// TwinCAT 3 PLC project PLC
// ProgramVersion: 3.1.4026.19
// libraries:
//   SPT Base Types, * (Beckhoff Automation LLC)
//   SPT Components, * (Beckhoff Automation LLC)
//   SPT Diagnostic, * (Beckhoff Automation LLC)
//   SPT EtherCat, * (Beckhoff Automation LLC)
//   SPT Event Logger, * (Beckhoff Automation LLC)
//   SPT Motion Control, * (Beckhoff Automation LLC)
//   SPT Utilities, * (Beckhoff Automation LLC)
//   Tc2_MC2, * (Beckhoff Automation GmbH)
//   Tc2_MC2_Camming, * (Beckhoff Automation GmbH)
//   Tc2_Standard, * (Beckhoff Automation GmbH)
//   Tc2_System, * (Beckhoff Automation GmbH)
//   Tc3_EventLogger, * (Beckhoff Automation GmbH)
//   Tc3_Module, * (Beckhoff Automation GmbH)
//   Tc3_PackML_V3, * (Beckhoff Automation GmbH)
// project tree:
//   / GlobalTextList.TcGTLO, PlcTask.TcTTO, Visualization Manager.TcVMO (not stored)
//   Modules/00 Machine/ Machine.TcPOU
//   Modules/01 Cam Module Table Select/ CamModule_TableSelect.TcPOU
//   Modules/01 Cam Module Table Select/DUTs/ ST_EM_Cfg_TableSelect.TcDUT, ST_EM_Cmd_TableSelect.TcDUT, ST_EM_HMI_TableSelect.TcDUT, ST_EM_Sts_TableSelect.TcDUT
//   Modules/02 Cam Module Update Table/ CamModule_UpdateTable.TcPOU
//   Modules/02 Cam Module Update Table/DUTs/ ST_EM_Cfg_UpdateTable.TcDUT, ST_EM_Cmd_UpdateTable.TcDUT, ST_EM_HMI_UpdateTable.TcDUT, ST_EM_Sts_UpdateTable.TcDUT
//   POUs/ MAIN.TcPOU
//   VISUs/ Visualization.TcVIS
// real-time tasks:
//   TASK PlcTask: cycle T#10ms, priority 20, ADS port 350
// motion (NC):
//   TASK NC-Task 1 SAF: cycle T#2ms, priority 4, ADS port 501
//   TASK NC-Task 1 SVB: cycle T#10ms, priority 8, ADS port 511
//   AXIS Cam Shaft Table Select (id 1)
//     OtherSettings: AllowMotionCmdToSlave=true
//     encoder EncType=1
//     drive DrvType=5
//       Analog: TorqueSetpointScale=10, ScaleFactorActTorque=0.1
//       TimeComp: TaskDelayCycles=1
//     controller CtrType=1
//       CtrPara: PriorControlFactor=1
//         Observer: BandWidth=20
//   AXIS Cam Follower Table Select (id 2)
//     OtherSettings: AllowMotionCmdToSlave=true
//     encoder EncType=1
//     drive DrvType=5
//       Analog: TorqueSetpointScale=10, ScaleFactorActTorque=0.1
//       TimeComp: TaskDelayCycles=1
//     controller CtrType=1
//       CtrPara: PriorControlFactor=1
//         Observer: BandWidth=20
//   AXIS Cam Shaft Update Table (id 3)
//     General: UnitFlags=#x00000004
//     OtherSettings: AllowMotionCmdToSlave=true
//     encoder EncType=1
//     drive DrvType=5
//       Analog: TorqueSetpointScale=10, ScaleFactorActTorque=0.1
//       TimeComp: TaskDelayCycles=1
//     controller CtrType=1
//       CtrPara: PriorControlFactor=1
//         Observer: BandWidth=20
//   AXIS Cam Follwer Update Table (id 4)
//     OtherSettings: AllowMotionCmdToSlave=true
//     encoder EncType=1
//     drive DrvType=5
//       Analog: TorqueSetpointScale=10, ScaleFactorActTorque=0.1
//     controller CtrType=1
//       CtrPara: PriorControlFactor=1
//         Observer: BandWidth=20
// variable links:
//   PLC/PLC Instance <-> NC-Task 1 SAF/Axes/Cam Follower Table Select
//     PlcTask Inputs/MAIN.Machine.CamModule_TableSelect.CamFollower.CamSlaveAxis._Axis.NcToPlc <-> Outputs/ToPlc
//     PlcTask Outputs/MAIN.Machine.CamModule_TableSelect.CamFollower.CamSlaveAxis._Axis.PlcToNc <-> Inputs/FromPlc
//   PLC/PLC Instance <-> NC-Task 1 SAF/Axes/Cam Follwer Update Table
//     PlcTask Inputs/MAIN.Machine.CamModule_UpdateTable.CamFollower.CamSlaveAxis._Axis.NcToPlc <-> Outputs/ToPlc
//     PlcTask Outputs/MAIN.Machine.CamModule_UpdateTable.CamFollower.CamSlaveAxis._Axis.PlcToNc <-> Inputs/FromPlc
//   PLC/PLC Instance <-> NC-Task 1 SAF/Axes/Cam Shaft Table Select
//     PlcTask Inputs/MAIN.Machine.CamModule_TableSelect.CamShaft.BasicAxis._Axis.NcToPlc <-> Outputs/ToPlc
//     PlcTask Outputs/MAIN.Machine.CamModule_TableSelect.CamShaft.BasicAxis._Axis.PlcToNc <-> Inputs/FromPlc
//   PLC/PLC Instance <-> NC-Task 1 SAF/Axes/Cam Shaft Update Table
//     PlcTask Inputs/MAIN.Machine.CamModule_UpdateTable.CamShaft.BasicAxis._Axis.NcToPlc <-> Outputs/ToPlc
//     PlcTask Outputs/MAIN.Machine.CamModule_UpdateTable.CamShaft.BasicAxis._Axis.PlcToNc <-> Inputs/FromPlc

CONFIGURATION PLC
    RESOURCE PLC ON TwinCAT3
        TASK PlcTask(INTERVAL := T#10ms, PRIORITY := 20);
        PROGRAM MAIN WITH PlcTask : MAIN;
    END_RESOURCE
END_CONFIGURATION

// ---- Modules/01 Cam Module Table Select/DUTs/ST_EM_Cfg_TableSelect.TcDUT
TYPE ST_EM_Cfg_TableSelect :
	STRUCT
		CamActivationMode : INT;
	END_STRUCT
END_TYPE

// ---- Modules/01 Cam Module Table Select/DUTs/ST_EM_Cmd_TableSelect.TcDUT
TYPE ST_EM_Cmd_TableSelect :
	STRUCT
		ChangeTable : BOOL;
		ChangeMode	: BOOL;
	END_STRUCT
END_TYPE

// ---- Modules/01 Cam Module Table Select/DUTs/ST_EM_HMI_TableSelect.TcDUT
TYPE ST_EM_HMI_TableSelect :
	STRUCT
		Cmd : ST_EM_Cmd_TableSelect;
		Cfg : ST_EM_Cfg_TableSelect;
		Sts : ST_EM_Sts_TableSelect;
	END_STRUCT
END_TYPE

// ---- Modules/01 Cam Module Table Select/DUTs/ST_EM_Sts_TableSelect.TcDUT
TYPE ST_EM_Sts_TableSelect :
	STRUCT
		CurrentTable : UDINT;
	END_STRUCT
END_TYPE

// ---- Modules/02 Cam Module Update Table/DUTs/ST_EM_Cfg_UpdateTable.TcDUT
TYPE ST_EM_Cfg_UpdateTable :
	STRUCT
		CamActivationMode : INT;
	END_STRUCT
END_TYPE

// ---- Modules/02 Cam Module Update Table/DUTs/ST_EM_Cmd_UpdateTable.TcDUT
TYPE ST_EM_Cmd_UpdateTable :
	STRUCT
		ChangeTable : BOOL;
		ChangeMode	: BOOL;
	END_STRUCT
END_TYPE

// ---- Modules/02 Cam Module Update Table/DUTs/ST_EM_HMI_UpdateTable.TcDUT
TYPE ST_EM_HMI_UpdateTable :
	STRUCT
		Cmd : ST_EM_Cmd_UpdateTable;
		Cfg : ST_EM_Cfg_UpdateTable;
		Sts : ST_EM_Sts_UpdateTable;
	END_STRUCT
END_TYPE

// ---- Modules/02 Cam Module Update Table/DUTs/ST_EM_Sts_UpdateTable.TcDUT
TYPE ST_EM_Sts_UpdateTable :
	STRUCT
		CurrentTable : UDINT;
	END_STRUCT
END_TYPE

// ---- POUs/MAIN.TcPOU
PROGRAM MAIN
VAR
	Machine : Machine := (Name := 'Machine');
END_VAR

// All sample code provided by Beckhoff Automation LLC are for illustrative purposes only and are provided “as is” and without any warranties, express or implied. Actual implementations in applications will vary significantly. Beckhoff Automation LLC shall have no liability for, and does not waive any rights in relation to, any code samples that it provides or the use of such code samples for any purpose.

(*
	Each Equipment Module holds 2 Axes.
	The first is the Cam Shaft (Master Axis), and the second is the Cam Follwer that will follow the cam table as the Cam Shaft is mmoving.
	The Cam table data is first populated during the Initialize method.

	The default value for ActivationMode is MC_CAMACTIVATION_INSTANTANEOUS.
	In the Cyclic Logic method the ActivationMode can be changed to:
	MC_CamActivationMode.MC_CAMACTIVATION_INSTANTANEOUS
	MC_CamActivationMode.MC_CAMACTIVATION_NEXTCYCLE
	MC_CamActivationMode.MC_CAMACTIVATION_ASSOONASPOSSIBLE
	
	Cam Module Table Select creates 2 tables in the Initialize method.
	Table 1 and Table 2
	In the Execute method it is possible to switch between tables based on the ActivationMode.
	
	Cam Module Update Table creates a single table in the Initialize method.
	In the Execute method the TableID is changed, the WriteParameters_1 or _2 is called to populate the new data, and the the UpdateTable() method is called.
	This process will continue to use the same table, but use the new values provided.

	The Visu provides the functionality to update the the running table based on the tables defined within the CamParameters.CamTable array.


*)

// For Debug Only
_AppInfo.KeepOutputsOnBP := TRUE;

//
Machine.CyclicLogic();

END_PROGRAM

// ---- Modules/00 Machine/Machine.TcPOU
FUNCTION_BLOCK Machine EXTENDS FB_PackML_BaseModule
VAR
	CamModule_TableSelect : CamModule_TableSelect := (Name := 'Cam Module Table Select');
	CamModule_UpdateTable : CamModule_UpdateTable := (Name := 'Cam Module Update Table');
END_VAR

// Automatically enables and disables HMI control based on the PackML mode
METHOD PROTECTED HMIPermissions

// This method is called cyclically by CyclicLogic()
AllowHMIControl(TRUE);
END_METHOD

// Basic module initialization logic
METHOD PROTECTED Initialize : BOOL;

// This method is called by CyclicLogic() as required
Initialize := FALSE;
CASE DescendantSequenceState OF
	0:
		RegisterSubmodule(SubModule := CamModule_TableSelect);
		RegisterSubmodule(SubModule := CamModule_UpdateTable);
		DescendantSequenceState := DescendantSequenceState + 10;

	10:
		IF SUPER^.Initialize() THEN
			Initialize := TRUE;
		END_IF
END_CASE
END_METHOD

END_FUNCTION_BLOCK

// ---- Modules/01 Cam Module Table Select/CamModule_TableSelect.TcPOU
FUNCTION_BLOCK CamModule_TableSelect EXTENDS FB_PackML_BaseModule
VAR
	CamShaft	  : FB_Component_BasicAxis	  := (Name := 'Cam Shaft');
	CamFollower	  : FB_Component_CamSlaveAxis := (Name := 'Cam Follower');
	CamParameters : ST_CamParameters;
	HMI			  : ST_EM_HMI_TableSelect;
END_VAR

METHOD PROTECTED Aborting
VAR
	CamShaftStop	: BOOL;
	CamFollowerStop : BOOL;
END_VAR
// Mode is ignored
CASE SequenceState OF
	0:
		NoStateTasksToComplete := FALSE;
		SequenceState		   := SequenceState + 10;

		// Setting Override to 100 will ensure velocity calculations are not limited
		CamShaft.Override	 := 100;
		CamFollower.Override := 100;

		// The below code is used to call the stop method of each axis while still in State 0, this is done for efficeniceny while aborting.

		// Stop all Axes
		CamShaftStop	:= CamShaft.Stop() OR CamShaft.Error;
		CamFollowerStop := CamFollower.Stop() OR CamFollower.Error;
		IF CamShaftStop AND CamFollowerStop THEN
			SequenceState := SequenceState + 10;
		END_IF

	10:
		IF CamShaft.Stopped AND CamFollower.Stopped THEN
			SequenceState := SequenceState + 10;
		END_IF

	20: // Disable Axis
		IF CamShaft.Disable() THEN
			SequenceState := SequenceState + 10;
		END_IF

	30:
		IF CamFollower.Disable() THEN
			SequenceState := SequenceState + 10;
		END_IF

	40:
		IF NOT CamShaft.Enabled AND NOT CamFollower.Enabled THEN
			SequenceState := SequenceState + 10;
		END_IF

	50:
		StateTasksComplete := TRUE;
END_CASE

SUPER^.Aborting();
END_METHOD

// This method contains code which will execute when this PackML module is in the Clearing state
METHOD PROTECTED Clearing

// Note: The Clear command can also be thought of as a fault reset depite the ambiguity in the naming of the Reset state. 

// This method is called as required by StateControl()
// Mode is ignored
CASE SequenceState OF
	0:
		NoStateTasksToComplete := FALSE;
		SequenceState		   := SequenceState + 10;

	10: // Reset Axis if Error
		IF CamShaft.Error THEN
			IF CamShaft.Reset() THEN
				SequenceState := SequenceState + 10;
			END_IF
		ELSE
			SequenceState := SequenceState + 10;
		END_IF

	20:
		IF CamFollower.InSync THEN
			IF CamFollower.Stop() THEN // This is used to decouple the axis
				SequenceState := SequenceState + 10;
			END_IF
		ELSE
			SequenceState := SequenceState + 10;
		END_IF

	30:
		IF CamFollower.Error THEN
			IF CamFollower.Reset() THEN
				SequenceState := SequenceState + 10;
			END_IF
		ELSE
			SequenceState := SequenceState + 10;
		END_IF

	40:
		StateTasksComplete := TRUE;
END_CASE

SUPER^.Clearing();
END_METHOD

METHOD PROTECTED Completing
CASE SequenceState OF
	0:
		NoStateTasksToComplete := FALSE;
		SequenceState		   := SequenceState + 10;

	10:
		IF CamShaft.Stop() THEN // This will also GearOut
			SequenceState := SequenceState + 10;
		END_IF

	20:
		IF CamFollower.Stop() THEN // This will also GearOut
			SequenceState := SequenceState + 10;
		END_IF

	30:
		IF CamShaft.Stopped AND CamFollower.Stopped THEN
			SequenceState := SequenceState + 10;
		END_IF

	40:
		StateTasksComplete := TRUE;
END_CASE

SUPER^.Completing();
END_METHOD

// This method serves as the entry point for all underlying FB logic

// This method should be called cyclically by descendant function blocks by invoking SUPER^.CyclicLogic().  Alternatively, the contents of this method could be reimplemented entirely in which case a call to this method would not be necessary.
METHOD PUBLIC CyclicLogic
IF NOT _InitComplete THEN
	_InitComplete := Initialize();
	RETURN;
END_IF

// HMI Status Update
HMI.Sts.CurrentTable := CamFollower.RunningTable;

// Change Activation Mode
IF HMI.Cmd.ChangeMode THEN
	CASE HMI.Cfg.CamActivationMode OF
		0:
			CamParameters.ChangeOptions.ActivationMode := MC_CamActivationMode.MC_CAMACTIVATION_INSTANTANEOUS;

		1:
			CamParameters.ChangeOptions.ActivationMode := MC_CamActivationMode.MC_CAMACTIVATION_NEXTCYCLE;

		2:
			CamParameters.ChangeOptions.ActivationMode := MC_CamActivationMode.MC_CAMACTIVATION_ASSOONASPOSSIBLE;
	END_CASE

	IF CamFollower.ChangeMode() THEN
		HMI.Cmd.ChangeMode := FALSE;
	END_IF
END_IF

SUPER^.CyclicLogic();
END_METHOD

// This method contains code which will execute when this PackML module is in the Execute state
METHOD PROTECTED Execute

(*
The base implementation of this method is empty. User must override this method to provide functionality.
This method is called as required by StateControl()
*)
CASE _CurrentMode OF
	E_PMLUnitMode.Production:
		CASE SequenceState OF
			0: // Start Cam Shaft
				IF CamShaft.MoveVelocity(50.0, FALSE) THEN
					SequenceState := SequenceState + 10;
				END_IF

			10: // Checking that the Cam Shaft is near the commanded speed 
				IF (CamShaft.ActualVelocity > (CamShaft.SetVelocity * 0.9)) THEN
					SequenceState := SequenceState + 10;
				END_IF

			20:
				IF HMI.Cmd.ChangeTable THEN
					HMI.Cmd.ChangeTable := FALSE;
					CASE CamFollower.RunningTable OF
						1:
							CamFollower.CamParameters.TableSelect := 2;

						2:
							CamFollower.CamParameters.TableSelect := 1;
					END_CASE

					SequenceState := SequenceState + 10;
				END_IF

			30:
				IF CamFollower.RunningTable = CamFollower.CamParameters.TableSelect THEN
					SequenceState := 20;
				END_IF;
		END_CASE
END_CASE
END_METHOD

// Basic module initialization logic
METHOD PROTECTED Initialize : BOOL;

// This method is called by CyclicLogic() as required
Initialize := FALSE;
CASE DescendantSequenceState OF
	0:
		RegisterComponent(Component := CamShaft);
		RegisterComponent(Component := CamFollower);
		DescendantSequenceState := DescendantSequenceState + 10;

	10:
		IF SUPER^.Initialize() THEN
			DescendantSequenceState := DescendantSequenceState + 10;
		END_IF

	20:
		// Create the Cam table data and store in CamParameters
		WriteCamParameters();

		// Set the Reference for the Axis Cam Parameters to the CamParameters
		CamFollower.CamParameters REF= CamParameters;

		// Setting the Reference of the FB_Component_CamSlaveAxis must be done after the component has been initialized
		CamFollower.Master REF= CamShaft.Axis;

		//
		DescendantSequenceState := DescendantSequenceState + 10;

	30:
		Initialize := TRUE;
END_CASE
END_METHOD

METHOD PROTECTED Starting
CASE _CommandedMode OF
	E_PMLUnitMode.Production:
		CASE SequenceState OF
			0:
				NoStateTasksToComplete := FALSE;
				SequenceState		   := SequenceState + 10;

			10: // Enable Axis 
				IF CamShaft.Enable() THEN
					SequenceState := SequenceState + 10;
				END_IF

			20:
				IF CamShaft.Enabled THEN
					SequenceState := SequenceState + 10;
				END_IF

			30: // This step is not required, but is used in this demo to ensure the CamShaft starts at 0
				IF CamShaft.MoveModulo(0.0, MC_Direction.MC_Shortest_Way, 0) THEN
					SequenceState := SequenceState + 10;
				END_IF

			40:
				IF NOT CamShaft.Busy THEN
					IF NOT CamShaft.Error THEN
						SequenceState := SequenceState + 10;
					END_IF
				END_IF

			50: // Enable Axis
				IF CamFollower.Enable() THEN
					SequenceState := SequenceState + 10;
				END_IF

			60:
				IF CamFollower.Enabled THEN
					SequenceState := SequenceState + 10;
				END_IF

			70: // This step is not required, but is used in the demo to ensure the follower starts at 0
				IF CamFollower.MoveAbsolute(0, 0) THEN
					SequenceState := SequenceState + 10;
				END_IF

			80:
				IF NOT CamFollower.Busy THEN
					IF NOT CamFollower.Error THEN
						SequenceState := SequenceState + 10;
					END_IF
				END_IF

			90: // Verify the Master axis is ready 
				IF CamFollower.Master.Status.Operational THEN
					SequenceState := SequenceState + 10;
				END_IF

			100: // Select the Cam Table to be used
				CamFollower.CamParameters.TableSelect := 1;
				SequenceState						  := SequenceState + 10;

			110: // Couple to Cam table with Master axis
				IF CamFollower.WaitingForCommand THEN
					IF CamFollower.StartSync() THEN // The Start Sync command will move the axes tho the necessary positions and then CamIn
						SequenceState := SequenceState + 10;
					END_IF
				END_IF

			120:
				IF CamFollower.InSync THEN
					SequenceState := SequenceState + 10;
				END_IF

			130:
				StateTasksComplete := TRUE;
		END_CASE
END_CASE

SUPER^.Starting();
END_METHOD

METHOD PROTECTED Stopping
CASE SequenceState OF
	0:
		NoStateTasksToComplete := FALSE;
		SequenceState		   := SequenceState + 10;

	10:
		IF CamShaft.Stop() THEN // This will also GearOut 
			SequenceState := SequenceState + 10;
		END_IF

	20:
		IF CamFollower.Stop() THEN // This will also GearOut  
			SequenceState := SequenceState + 10;
		END_IF

	30:
		IF CamShaft.Stopped AND CamFollower.Stopped THEN
			SequenceState := SequenceState + 10;
		END_IF

	40:
		StateTasksComplete := TRUE;
END_CASE

SUPER^.Stopping();
END_METHOD

METHOD WriteCamParameters
VAR
	PointIdx : UDINT;
	i		 : UDINT;
	Start	 : UDINT;
END_VAR
// Table 1 Data
CamParameters.CamTableId										:= CamShaft.Axis.NcToPlc.AxisId;
CamParameters.CamTable[CamParameters.CamTableId].NumberOfPoints := Parameters_MotionControl.CAM_SLAVE_AXIS_MAX_CAM_POINTS;
PointIdx														:= 0;

//
PointIdx																			:= PointIdx + 1;
CamParameters.CamTable[CamParameters.CamTableId].Points[PointIdx].PointIndex		:= PointIdx;
CamParameters.CamTable[CamParameters.CamTableId].Points[PointIdx].FunctionType		:= MC_MotionFunctionType.MOTIONFUNCTYPE_POLYNOM5;
CamParameters.CamTable[CamParameters.CamTableId].Points[PointIdx].PointType			:= MC_MotionPointType.MOTIONPOINTTYPE_REST;
CamParameters.CamTable[CamParameters.CamTableId].Points[PointIdx].RelIndexNextPoint := 1;
CamParameters.CamTable[CamParameters.CamTableId].Points[PointIdx].MasterPos			:= 0.0;
CamParameters.CamTable[CamParameters.CamTableId].Points[PointIdx].SlavePos			:= 0.0;

//
PointIdx																			:= PointIdx + 1;
CamParameters.CamTable[CamParameters.CamTableId].Points[PointIdx].PointIndex		:= PointIdx;
CamParameters.CamTable[CamParameters.CamTableId].Points[PointIdx].FunctionType		:= MC_MotionFunctionType.MOTIONFUNCTYPE_POLYNOM5;
CamParameters.CamTable[CamParameters.CamTableId].Points[PointIdx].PointType			:= MC_MotionPointType.MOTIONPOINTTYPE_VELOCITY;
CamParameters.CamTable[CamParameters.CamTableId].Points[PointIdx].RelIndexNextPoint := 1;
CamParameters.CamTable[CamParameters.CamTableId].Points[PointIdx].MasterPos			:= 90.0;
CamParameters.CamTable[CamParameters.CamTableId].Points[PointIdx].SlavePos			:= 0.0;

//
PointIdx																			:= PointIdx + 1;
CamParameters.CamTable[CamParameters.CamTableId].Points[PointIdx].PointIndex		:= PointIdx;
CamParameters.CamTable[CamParameters.CamTableId].Points[PointIdx].FunctionType		:= MC_MotionFunctionType.MOTIONFUNCTYPE_POLYNOM5;
CamParameters.CamTable[CamParameters.CamTableId].Points[PointIdx].PointType			:= MC_MotionPointType.MOTIONPOINTTYPE_VELOCITY;
CamParameters.CamTable[CamParameters.CamTableId].Points[PointIdx].RelIndexNextPoint := 1;
CamParameters.CamTable[CamParameters.CamTableId].Points[PointIdx].MasterPos			:= 180.0;
CamParameters.CamTable[CamParameters.CamTableId].Points[PointIdx].SlavePos			:= 10.0;

//
PointIdx																			:= PointIdx + 1;
CamParameters.CamTable[CamParameters.CamTableId].Points[PointIdx].PointIndex		:= PointIdx;
CamParameters.CamTable[CamParameters.CamTableId].Points[PointIdx].FunctionType		:= MC_MotionFunctionType.MOTIONFUNCTYPE_POLYNOM5;
CamParameters.CamTable[CamParameters.CamTableId].Points[PointIdx].PointType			:= MC_MotionPointType.MOTIONPOINTTYPE_VELOCITY;
CamParameters.CamTable[CamParameters.CamTableId].Points[PointIdx].RelIndexNextPoint := 1;
CamParameters.CamTable[CamParameters.CamTableId].Points[PointIdx].MasterPos			:= 270.0;
CamParameters.CamTable[CamParameters.CamTableId].Points[PointIdx].SlavePos			:= 10.0;

//
PointIdx																			:= PointIdx + 1;
CamParameters.CamTable[CamParameters.CamTableId].Points[PointIdx].PointIndex		:= PointIdx;
CamParameters.CamTable[CamParameters.CamTableId].Points[PointIdx].FunctionType		:= MC_MotionFunctionType.MOTIONFUNCTYPE_POLYNOM5;
CamParameters.CamTable[CamParameters.CamTableId].Points[PointIdx].PointType			:= MC_MotionPointType.MOTIONPOINTTYPE_VELOCITY;
CamParameters.CamTable[CamParameters.CamTableId].Points[PointIdx].RelIndexNextPoint := 1;
CamParameters.CamTable[CamParameters.CamTableId].Points[PointIdx].MasterPos			:= 360.0;
CamParameters.CamTable[CamParameters.CamTableId].Points[PointIdx].SlavePos			:= 0.0;

// Fill the rest of the table with ignore points
Start := PointIdx + 1;
FOR PointIdx := Start TO Parameters_MotionControl.CAM_SLAVE_AXIS_MAX_CAM_POINTS DO
	CamParameters.CamTable[CamParameters.CamTableId].Points[PointIdx].PointIndex		:= PointIdx;
	CamParameters.CamTable[CamParameters.CamTableId].Points[PointIdx].FunctionType		:= MC_MotionFunctionType.MOTIONFUNCTYPE_NOTDEF;
	CamParameters.CamTable[CamParameters.CamTableId].Points[PointIdx].PointType			:= MC_MotionPointType.MOTIONPOINTTYPE_IGNORE;
	CamParameters.CamTable[CamParameters.CamTableId].Points[PointIdx].RelIndexNextPoint := 1;
	CamParameters.CamTable[CamParameters.CamTableId].Points[PointIdx].MasterPos			:= 0.0;
	CamParameters.CamTable[CamParameters.CamTableId].Points[PointIdx].SlavePos			:= 0.0;
END_FOR

// Set Lasst Point RelNext to 0
CamParameters.CamTable[CamParameters.CamTableId].Points[Parameters_MotionControl.CAM_SLAVE_AXIS_MAX_CAM_POINTS].RelIndexNextPoint := 0;

// Table 2 Data
CamParameters.CamTableId										:= CamShaft.Axis.NcToPlc.AxisId + 1;
CamParameters.CamTable[CamParameters.CamTableId].NumberOfPoints := Parameters_MotionControl.CAM_SLAVE_AXIS_MAX_CAM_POINTS;
PointIdx														:= 0;

//
PointIdx																			:= PointIdx + 1;
CamParameters.CamTable[CamParameters.CamTableId].Points[PointIdx].PointIndex		:= PointIdx;
CamParameters.CamTable[CamParameters.CamTableId].Points[PointIdx].FunctionType		:= MC_MotionFunctionType.MOTIONFUNCTYPE_POLYNOM5;
CamParameters.CamTable[CamParameters.CamTableId].Points[PointIdx].PointType			:= MC_MotionPointType.MOTIONPOINTTYPE_REST;
CamParameters.CamTable[CamParameters.CamTableId].Points[PointIdx].RelIndexNextPoint := 1;
CamParameters.CamTable[CamParameters.CamTableId].Points[PointIdx].MasterPos			:= 0.0;
CamParameters.CamTable[CamParameters.CamTableId].Points[PointIdx].SlavePos			:= 0.0;

//
PointIdx																			:= PointIdx + 1;
CamParameters.CamTable[CamParameters.CamTableId].Points[PointIdx].PointIndex		:= PointIdx;
CamParameters.CamTable[CamParameters.CamTableId].Points[PointIdx].FunctionType		:= MC_MotionFunctionType.MOTIONFUNCTYPE_POLYNOM5;
CamParameters.CamTable[CamParameters.CamTableId].Points[PointIdx].PointType			:= MC_MotionPointType.MOTIONPOINTTYPE_VELOCITY;
CamParameters.CamTable[CamParameters.CamTableId].Points[PointIdx].RelIndexNextPoint := 1;
CamParameters.CamTable[CamParameters.CamTableId].Points[PointIdx].MasterPos			:= 90.0;
CamParameters.CamTable[CamParameters.CamTableId].Points[PointIdx].SlavePos			:= 0.0;

//
PointIdx																			:= PointIdx + 1;
CamParameters.CamTable[CamParameters.CamTableId].Points[PointIdx].PointIndex		:= PointIdx;
CamParameters.CamTable[CamParameters.CamTableId].Points[PointIdx].FunctionType		:= MC_MotionFunctionType.MOTIONFUNCTYPE_POLYNOM5;
CamParameters.CamTable[CamParameters.CamTableId].Points[PointIdx].PointType			:= MC_MotionPointType.MOTIONPOINTTYPE_VELOCITY;
CamParameters.CamTable[CamParameters.CamTableId].Points[PointIdx].RelIndexNextPoint := 1;
CamParameters.CamTable[CamParameters.CamTableId].Points[PointIdx].MasterPos			:= 180.0;
CamParameters.CamTable[CamParameters.CamTableId].Points[PointIdx].SlavePos			:= 20.0;

//
PointIdx																			:= PointIdx + 1;
CamParameters.CamTable[CamParameters.CamTableId].Points[PointIdx].PointIndex		:= PointIdx;
CamParameters.CamTable[CamParameters.CamTableId].Points[PointIdx].FunctionType		:= MC_MotionFunctionType.MOTIONFUNCTYPE_POLYNOM5;
CamParameters.CamTable[CamParameters.CamTableId].Points[PointIdx].PointType			:= MC_MotionPointType.MOTIONPOINTTYPE_REST;
CamParameters.CamTable[CamParameters.CamTableId].Points[PointIdx].RelIndexNextPoint := 1;
CamParameters.CamTable[CamParameters.CamTableId].Points[PointIdx].MasterPos			:= 270.0;
CamParameters.CamTable[CamParameters.CamTableId].Points[PointIdx].SlavePos			:= 20.0;

//
PointIdx																			:= PointIdx + 1;
CamParameters.CamTable[CamParameters.CamTableId].Points[PointIdx].PointIndex		:= PointIdx;
CamParameters.CamTable[CamParameters.CamTableId].Points[PointIdx].FunctionType		:= MC_MotionFunctionType.MOTIONFUNCTYPE_POLYNOM5;
CamParameters.CamTable[CamParameters.CamTableId].Points[PointIdx].PointType			:= MC_MotionPointType.MOTIONPOINTTYPE_REST;
CamParameters.CamTable[CamParameters.CamTableId].Points[PointIdx].RelIndexNextPoint := 1;
CamParameters.CamTable[CamParameters.CamTableId].Points[PointIdx].MasterPos			:= 360.0;
CamParameters.CamTable[CamParameters.CamTableId].Points[PointIdx].SlavePos			:= 0.0;

// Fill the rest of the table with ignore points
Start := PointIdx + 1;
FOR PointIdx := Start TO Parameters_MotionControl.CAM_SLAVE_AXIS_MAX_CAM_POINTS DO
	CamParameters.CamTable[CamParameters.CamTableId].Points[PointIdx].PointIndex		:= PointIdx;
	CamParameters.CamTable[CamParameters.CamTableId].Points[PointIdx].FunctionType		:= MC_MotionFunctionType.MOTIONFUNCTYPE_NOTDEF;
	CamParameters.CamTable[CamParameters.CamTableId].Points[PointIdx].PointType			:= MC_MotionPointType.MOTIONPOINTTYPE_IGNORE;
	CamParameters.CamTable[CamParameters.CamTableId].Points[PointIdx].RelIndexNextPoint := 1;
	CamParameters.CamTable[CamParameters.CamTableId].Points[PointIdx].MasterPos			:= 0.0;
	CamParameters.CamTable[CamParameters.CamTableId].Points[PointIdx].SlavePos			:= 0.0;
END_FOR

// Set Lasst Point RelNext to 0
CamParameters.CamTable[CamParameters.CamTableId].Points[Parameters_MotionControl.CAM_SLAVE_AXIS_MAX_CAM_POINTS].RelIndexNextPoint := 0;
END_METHOD

END_FUNCTION_BLOCK

// ---- Modules/02 Cam Module Update Table/CamModule_UpdateTable.TcPOU
FUNCTION_BLOCK CamModule_UpdateTable EXTENDS FB_PackML_BaseModule
VAR
	CamShaft	  : FB_Component_BasicAxis	  := (Name := 'Cam Shaft');
	CamFollower	  : FB_Component_CamSlaveAxis := (Name := 'Cam Follower');
	CamParameters : ST_CamParameters;
	HMI			  : ST_EM_HMI_UpdateTable;
	_NextTable	  : INT;
END_VAR

METHOD PROTECTED Aborting
VAR
	CamShaftStop	: BOOL;
	CamFollowerStop : BOOL;
END_VAR
// Mode is ignored
CASE SequenceState OF
	0:
		NoStateTasksToComplete := FALSE;
		SequenceState		   := SequenceState + 10;

		// Setting Override to 100 will ensure velocity calculations are not limited
		CamShaft.Override	 := 100;
		CamFollower.Override := 100;

		// The below code is used to call the stop method of each axis while still in State 0, this is done for efficeniceny while aborting.

		// Stop all Axes
		CamShaftStop	:= CamShaft.Stop() OR CamShaft.Error;
		CamFollowerStop := CamFollower.Stop() OR CamFollower.Error;
		IF CamShaftStop AND CamFollowerStop THEN
			SequenceState := SequenceState + 10;
		END_IF

	10:
		IF CamShaft.Stopped AND CamFollower.Stopped THEN
			SequenceState := SequenceState + 10;
		END_IF

	20: // Disable Axis
		IF CamShaft.Disable() THEN
			SequenceState := SequenceState + 10;
		END_IF

	30:
		IF CamFollower.Disable() THEN
			SequenceState := SequenceState + 10;
		END_IF

	40:
		IF NOT CamShaft.Enabled AND NOT CamFollower.Enabled THEN
			SequenceState := SequenceState + 10;
		END_IF

	50:
		StateTasksComplete := TRUE;
END_CASE

SUPER^.Aborting();
END_METHOD

// This method contains code which will execute when this PackML module is in the Clearing state
METHOD PROTECTED Clearing

// Note: The Clear command can also be thought of as a fault reset depite the ambiguity in the naming of the Reset state. 

// This method is called as required by StateControl()
// Mode is ignored
CASE SequenceState OF
	0:
		NoStateTasksToComplete := FALSE;
		SequenceState		   := SequenceState + 10;

	10: // Reset Axis if Error
		IF CamShaft.Error THEN
			IF CamShaft.Reset() THEN
				SequenceState := SequenceState + 10;
			END_IF
		ELSE
			SequenceState := SequenceState + 10;
		END_IF

	20:
		IF CamFollower.InSync THEN
			IF CamFollower.Stop() THEN // This is used to decouple the axis
				SequenceState := SequenceState + 10;
			END_IF
		ELSE
			SequenceState := SequenceState + 10;
		END_IF

	30:
		IF CamFollower.Error THEN
			IF CamFollower.Reset() THEN
				SequenceState := SequenceState + 10;
			END_IF
		ELSE
			SequenceState := SequenceState + 10;
		END_IF

	40:
		StateTasksComplete := TRUE;
END_CASE

SUPER^.Clearing();
END_METHOD

METHOD PROTECTED Completing
CASE SequenceState OF
	0:
		NoStateTasksToComplete := FALSE;
		SequenceState		   := SequenceState + 10;

	10:
		IF CamShaft.Stop() THEN // This will also GearOut
			SequenceState := SequenceState + 10;
		END_IF

	20:
		IF CamFollower.Stop() THEN // This will also GearOut
			SequenceState := SequenceState + 10;
		END_IF

	30:
		IF CamShaft.Stopped AND CamFollower.Stopped THEN
			SequenceState := SequenceState + 10;
		END_IF

	40:
		StateTasksComplete := TRUE;
END_CASE

SUPER^.Completing();
END_METHOD

// This method serves as the entry point for all underlying FB logic

// This method should be called cyclically by descendant function blocks by invoking SUPER^.CyclicLogic().  Alternatively, the contents of this method could be reimplemented entirely in which case a call to this method would not be necessary.
METHOD PUBLIC CyclicLogic
IF NOT _InitComplete THEN
	_InitComplete := Initialize();
	RETURN;
END_IF

// HMI Status Update
HMI.Sts.CurrentTable := CamFollower.RunningTable;

// Change Activation Mode
IF HMI.Cmd.ChangeMode THEN
	CASE HMI.Cfg.CamActivationMode OF
		0:
			CamParameters.ChangeOptions.ActivationMode := MC_CamActivationMode.MC_CAMACTIVATION_INSTANTANEOUS;

		1:
			CamParameters.ChangeOptions.ActivationMode := MC_CamActivationMode.MC_CAMACTIVATION_NEXTCYCLE;

		2:
			CamParameters.ChangeOptions.ActivationMode := MC_CamActivationMode.MC_CAMACTIVATION_ASSOONASPOSSIBLE;
	END_CASE

	IF CamFollower.ChangeMode() THEN
		HMI.Cmd.ChangeMode := FALSE;
	END_IF
END_IF

SUPER^.CyclicLogic();
END_METHOD

// This method contains code which will execute when this PackML module is in the Execute state
METHOD PROTECTED Execute

(*
The base implementation of this method is empty. User must override this method to provide functionality.
This method is called as required by StateControl()
*)
CASE _CurrentMode OF
	E_PMLUnitMode.Production:
		CASE SequenceState OF
			0: // Start Cam Shaft
				IF CamShaft.MoveVelocity(50.0, FALSE) THEN
					SequenceState := SequenceState + 10;
				END_IF

			10: // Checking that the Cam Shaft is near the commanded speed 
				IF (CamShaft.ActualVelocity > (CamShaft.SetVelocity * 0.9)) THEN
					SequenceState := SequenceState + 10;
				END_IF

			20:
				IF HMI.Cmd.ChangeTable THEN
					HMI.Cmd.ChangeTable := FALSE;
					CASE _NextTable OF
						1:
							WriteCamParameters_2();
							CamFollower.UpdateTable();

						2:
							WriteCamParameters_1();
							CamFollower.UpdateTable();
					END_CASE

					SequenceState := SequenceState + 10;
				END_IF

			30:
				IF CamFollower.RunningTable = CamFollower.CamParameters.TableSelect THEN
					SequenceState := 20;
				END_IF;
		END_CASE
END_CASE
END_METHOD

// Basic module initialization logic
METHOD PROTECTED Initialize : BOOL;

// This method is called by CyclicLogic() as required
Initialize := FALSE;
CASE DescendantSequenceState OF
	0:
		RegisterComponent(Component := CamShaft);
		RegisterComponent(Component := CamFollower);
		DescendantSequenceState := DescendantSequenceState + 10;

	10:
		IF SUPER^.Initialize() THEN
			DescendantSequenceState := DescendantSequenceState + 10;
		END_IF

	20:
		// Create the Cam table data and store in CamParameters
		WriteCamParameters();

		// Set the Reference for the Axis Cam Parameters to the CamParameters
		CamFollower.CamParameters REF= CamParameters;

		// Setting the Reference of the FB_Component_CamSlaveAxis must be done after the component has been initialized
		CamFollower.Master REF= CamShaft.Axis;

		//
		DescendantSequenceState := DescendantSequenceState + 10;

	30:
		Initialize := TRUE;
END_CASE
END_METHOD

METHOD PROTECTED Starting
CASE _CommandedMode OF
	E_PMLUnitMode.Production:
		CASE SequenceState OF
			0:
				NoStateTasksToComplete := FALSE;
				SequenceState		   := SequenceState + 10;

			10: // Enable Axis 
				IF CamShaft.Enable() THEN
					SequenceState := SequenceState + 10;
				END_IF

			20:
				IF CamShaft.Enabled THEN
					SequenceState := SequenceState + 10;
				END_IF

			30: // This step is not required, but is used in this demo to ensure the CamShaft starts at 0
				IF CamShaft.MoveModulo(0.0, MC_Direction.MC_Shortest_Way, 0) THEN
					SequenceState := SequenceState + 10;
				END_IF

			40:
				IF NOT CamShaft.Busy THEN
					IF NOT CamShaft.Error THEN
						SequenceState := SequenceState + 10;
					END_IF
				END_IF

			50: // Enable Axis
				IF CamFollower.Enable() THEN
					SequenceState := SequenceState + 10;
				END_IF

			60:
				IF CamFollower.Enabled THEN
					SequenceState := SequenceState + 10;
				END_IF

			70: // This step is not required, but is used in the demo to ensure the follower starts at 0
				IF CamFollower.MoveAbsolute(0, 0) THEN
					SequenceState := SequenceState + 10;
				END_IF

			80:
				IF NOT CamFollower.Busy THEN
					IF NOT CamFollower.Error THEN
						SequenceState := SequenceState + 10;
					END_IF
				END_IF

			90: // Verify the Master axis is ready 
				IF CamFollower.Master.Status.Operational THEN
					SequenceState := SequenceState + 10;
				END_IF

			100: // Select the Cam Table to be used
				CamFollower.CamParameters.TableSelect := 3;
				SequenceState						  := SequenceState + 10;

			110: // Couple to Cam table with Master axis
				IF CamFollower.WaitingForCommand THEN
					IF CamFollower.StartSync() THEN // The Start Sync command will move the axes tho the necessary positions and then CamIn
						SequenceState := SequenceState + 10;
					END_IF
				END_IF

			120:
				IF CamFollower.InSync THEN
					SequenceState := SequenceState + 10;
				END_IF

			130:
				StateTasksComplete := TRUE;
		END_CASE
END_CASE

SUPER^.Starting();
END_METHOD

METHOD PROTECTED Stopping
CASE SequenceState OF
	0:
		NoStateTasksToComplete := FALSE;
		SequenceState		   := SequenceState + 10;

	10:
		IF CamShaft.Stop() THEN // This will also GearOut 
			SequenceState := SequenceState + 10;
		END_IF

	20:
		IF CamFollower.Stop() THEN // This will also GearOut  
			SequenceState := SequenceState + 10;
		END_IF

	30:
		IF CamShaft.Stopped AND CamFollower.Stopped THEN
			SequenceState := SequenceState + 10;
		END_IF

	40:
		StateTasksComplete := TRUE;
END_CASE

SUPER^.Stopping();
END_METHOD

METHOD WriteCamParameters
WriteCamParameters_1();
_NextTable := 1;
END_METHOD

METHOD WriteCamParameters_1
VAR
	PointIdx : UDINT;
	i		 : UDINT;
	Start	 : UDINT;
END_VAR
_NextTable := 1;

// Update Table 1 Data
CamParameters.CamTableId										:= CamShaft.Axis.NcToPlc.AxisId;
CamParameters.CamTable[CamParameters.CamTableId].NumberOfPoints := Parameters_MotionControl.CAM_SLAVE_AXIS_MAX_CAM_POINTS;
PointIdx														:= 0;

//
PointIdx																			:= PointIdx + 1;
CamParameters.CamTable[CamParameters.CamTableId].Points[PointIdx].PointIndex		:= PointIdx;
CamParameters.CamTable[CamParameters.CamTableId].Points[PointIdx].FunctionType		:= MC_MotionFunctionType.MOTIONFUNCTYPE_POLYNOM5;
CamParameters.CamTable[CamParameters.CamTableId].Points[PointIdx].PointType			:= MC_MotionPointType.MOTIONPOINTTYPE_REST;
CamParameters.CamTable[CamParameters.CamTableId].Points[PointIdx].RelIndexNextPoint := 1;
CamParameters.CamTable[CamParameters.CamTableId].Points[PointIdx].MasterPos			:= 0.0;
CamParameters.CamTable[CamParameters.CamTableId].Points[PointIdx].SlavePos			:= 0.0;

//
PointIdx																			:= PointIdx + 1;
CamParameters.CamTable[CamParameters.CamTableId].Points[PointIdx].PointIndex		:= PointIdx;
CamParameters.CamTable[CamParameters.CamTableId].Points[PointIdx].FunctionType		:= MC_MotionFunctionType.MOTIONFUNCTYPE_POLYNOM5;
CamParameters.CamTable[CamParameters.CamTableId].Points[PointIdx].PointType			:= MC_MotionPointType.MOTIONPOINTTYPE_VELOCITY;
CamParameters.CamTable[CamParameters.CamTableId].Points[PointIdx].RelIndexNextPoint := 1;
CamParameters.CamTable[CamParameters.CamTableId].Points[PointIdx].MasterPos			:= 90.0;
CamParameters.CamTable[CamParameters.CamTableId].Points[PointIdx].SlavePos			:= 0.0;

//
PointIdx																			:= PointIdx + 1;
CamParameters.CamTable[CamParameters.CamTableId].Points[PointIdx].PointIndex		:= PointIdx;
CamParameters.CamTable[CamParameters.CamTableId].Points[PointIdx].FunctionType		:= MC_MotionFunctionType.MOTIONFUNCTYPE_POLYNOM5;
CamParameters.CamTable[CamParameters.CamTableId].Points[PointIdx].PointType			:= MC_MotionPointType.MOTIONPOINTTYPE_VELOCITY;
CamParameters.CamTable[CamParameters.CamTableId].Points[PointIdx].RelIndexNextPoint := 1;
CamParameters.CamTable[CamParameters.CamTableId].Points[PointIdx].MasterPos			:= 180.0;
CamParameters.CamTable[CamParameters.CamTableId].Points[PointIdx].SlavePos			:= 10.0;

//
PointIdx																			:= PointIdx + 1;
CamParameters.CamTable[CamParameters.CamTableId].Points[PointIdx].PointIndex		:= PointIdx;
CamParameters.CamTable[CamParameters.CamTableId].Points[PointIdx].FunctionType		:= MC_MotionFunctionType.MOTIONFUNCTYPE_POLYNOM5;
CamParameters.CamTable[CamParameters.CamTableId].Points[PointIdx].PointType			:= MC_MotionPointType.MOTIONPOINTTYPE_REST;
CamParameters.CamTable[CamParameters.CamTableId].Points[PointIdx].RelIndexNextPoint := 1;
CamParameters.CamTable[CamParameters.CamTableId].Points[PointIdx].MasterPos			:= 270.0;
CamParameters.CamTable[CamParameters.CamTableId].Points[PointIdx].SlavePos			:= 10.0;

//
PointIdx																			:= PointIdx + 1;
CamParameters.CamTable[CamParameters.CamTableId].Points[PointIdx].PointIndex		:= PointIdx;
CamParameters.CamTable[CamParameters.CamTableId].Points[PointIdx].FunctionType		:= MC_MotionFunctionType.MOTIONFUNCTYPE_POLYNOM5;
CamParameters.CamTable[CamParameters.CamTableId].Points[PointIdx].PointType			:= MC_MotionPointType.MOTIONPOINTTYPE_REST;
CamParameters.CamTable[CamParameters.CamTableId].Points[PointIdx].RelIndexNextPoint := 1;
CamParameters.CamTable[CamParameters.CamTableId].Points[PointIdx].MasterPos			:= 360.0;
CamParameters.CamTable[CamParameters.CamTableId].Points[PointIdx].SlavePos			:= 0.0;

// Fill the rest of the table with ignore points
Start := PointIdx + 1;
FOR PointIdx := Start TO Parameters_MotionControl.CAM_SLAVE_AXIS_MAX_CAM_POINTS DO
	CamParameters.CamTable[CamParameters.CamTableId].Points[PointIdx].PointIndex		:= PointIdx;
	CamParameters.CamTable[CamParameters.CamTableId].Points[PointIdx].FunctionType		:= MC_MotionFunctionType.MOTIONFUNCTYPE_NOTDEF;
	CamParameters.CamTable[CamParameters.CamTableId].Points[PointIdx].PointType			:= MC_MotionPointType.MOTIONPOINTTYPE_IGNORE;
	CamParameters.CamTable[CamParameters.CamTableId].Points[PointIdx].RelIndexNextPoint := 1;
	CamParameters.CamTable[CamParameters.CamTableId].Points[PointIdx].MasterPos			:= 0.0;
	CamParameters.CamTable[CamParameters.CamTableId].Points[PointIdx].SlavePos			:= 0.0;
END_FOR

// Set Lasst Point RelNext to 0
CamParameters.CamTable[CamParameters.CamTableId].Points[Parameters_MotionControl.CAM_SLAVE_AXIS_MAX_CAM_POINTS].RelIndexNextPoint := 0;
END_METHOD

METHOD WriteCamParameters_2
VAR
	PointIdx : UDINT;
	i		 : UDINT;
	Start	 : UDINT;
END_VAR
_NextTable := 2;

// Update Table 1 Data
CamParameters.CamTableId										:= CamShaft.Axis.NcToPlc.AxisId;
CamParameters.CamTable[CamParameters.CamTableId].NumberOfPoints := Parameters_MotionControl.CAM_SLAVE_AXIS_MAX_CAM_POINTS;
PointIdx														:= 0;

//
PointIdx																			:= PointIdx + 1;
CamParameters.CamTable[CamParameters.CamTableId].Points[PointIdx].PointIndex		:= PointIdx;
CamParameters.CamTable[CamParameters.CamTableId].Points[PointIdx].FunctionType		:= MC_MotionFunctionType.MOTIONFUNCTYPE_POLYNOM5;
CamParameters.CamTable[CamParameters.CamTableId].Points[PointIdx].PointType			:= MC_MotionPointType.MOTIONPOINTTYPE_REST;
CamParameters.CamTable[CamParameters.CamTableId].Points[PointIdx].RelIndexNextPoint := 1;
CamParameters.CamTable[CamParameters.CamTableId].Points[PointIdx].MasterPos			:= 0.0;
CamParameters.CamTable[CamParameters.CamTableId].Points[PointIdx].SlavePos			:= 0.0;

//
PointIdx																			:= PointIdx + 1;
CamParameters.CamTable[CamParameters.CamTableId].Points[PointIdx].PointIndex		:= PointIdx;
CamParameters.CamTable[CamParameters.CamTableId].Points[PointIdx].FunctionType		:= MC_MotionFunctionType.MOTIONFUNCTYPE_POLYNOM5;
CamParameters.CamTable[CamParameters.CamTableId].Points[PointIdx].PointType			:= MC_MotionPointType.MOTIONPOINTTYPE_VELOCITY;
CamParameters.CamTable[CamParameters.CamTableId].Points[PointIdx].RelIndexNextPoint := 1;
CamParameters.CamTable[CamParameters.CamTableId].Points[PointIdx].MasterPos			:= 90.0;
CamParameters.CamTable[CamParameters.CamTableId].Points[PointIdx].SlavePos			:= 0.0;

//
PointIdx																			:= PointIdx + 1;
CamParameters.CamTable[CamParameters.CamTableId].Points[PointIdx].PointIndex		:= PointIdx;
CamParameters.CamTable[CamParameters.CamTableId].Points[PointIdx].FunctionType		:= MC_MotionFunctionType.MOTIONFUNCTYPE_POLYNOM5;
CamParameters.CamTable[CamParameters.CamTableId].Points[PointIdx].PointType			:= MC_MotionPointType.MOTIONPOINTTYPE_VELOCITY;
CamParameters.CamTable[CamParameters.CamTableId].Points[PointIdx].RelIndexNextPoint := 1;
CamParameters.CamTable[CamParameters.CamTableId].Points[PointIdx].MasterPos			:= 180.0;
CamParameters.CamTable[CamParameters.CamTableId].Points[PointIdx].SlavePos			:= 15.0;

//
PointIdx																			:= PointIdx + 1;
CamParameters.CamTable[CamParameters.CamTableId].Points[PointIdx].PointIndex		:= PointIdx;
CamParameters.CamTable[CamParameters.CamTableId].Points[PointIdx].FunctionType		:= MC_MotionFunctionType.MOTIONFUNCTYPE_POLYNOM5;
CamParameters.CamTable[CamParameters.CamTableId].Points[PointIdx].PointType			:= MC_MotionPointType.MOTIONPOINTTYPE_REST;
CamParameters.CamTable[CamParameters.CamTableId].Points[PointIdx].RelIndexNextPoint := 1;
CamParameters.CamTable[CamParameters.CamTableId].Points[PointIdx].MasterPos			:= 270.0;
CamParameters.CamTable[CamParameters.CamTableId].Points[PointIdx].SlavePos			:= 15.0;

//
PointIdx																			:= PointIdx + 1;
CamParameters.CamTable[CamParameters.CamTableId].Points[PointIdx].PointIndex		:= PointIdx;
CamParameters.CamTable[CamParameters.CamTableId].Points[PointIdx].FunctionType		:= MC_MotionFunctionType.MOTIONFUNCTYPE_POLYNOM5;
CamParameters.CamTable[CamParameters.CamTableId].Points[PointIdx].PointType			:= MC_MotionPointType.MOTIONPOINTTYPE_REST;
CamParameters.CamTable[CamParameters.CamTableId].Points[PointIdx].RelIndexNextPoint := 1;
CamParameters.CamTable[CamParameters.CamTableId].Points[PointIdx].MasterPos			:= 360.0;
CamParameters.CamTable[CamParameters.CamTableId].Points[PointIdx].SlavePos			:= 0.0;

// Fill the rest of the table with ignore points
Start := PointIdx + 1;
FOR PointIdx := Start TO Parameters_MotionControl.CAM_SLAVE_AXIS_MAX_CAM_POINTS DO
	CamParameters.CamTable[CamParameters.CamTableId].Points[PointIdx].PointIndex		:= PointIdx;
	CamParameters.CamTable[CamParameters.CamTableId].Points[PointIdx].FunctionType		:= MC_MotionFunctionType.MOTIONFUNCTYPE_NOTDEF;
	CamParameters.CamTable[CamParameters.CamTableId].Points[PointIdx].PointType			:= MC_MotionPointType.MOTIONPOINTTYPE_IGNORE;
	CamParameters.CamTable[CamParameters.CamTableId].Points[PointIdx].RelIndexNextPoint := 1;
	CamParameters.CamTable[CamParameters.CamTableId].Points[PointIdx].MasterPos			:= 0.0;
	CamParameters.CamTable[CamParameters.CamTableId].Points[PointIdx].SlavePos			:= 0.0;
END_FOR

// Set Lasst Point RelNext to 0
CamParameters.CamTable[CamParameters.CamTableId].Points[Parameters_MotionControl.CAM_SLAVE_AXIS_MAX_CAM_POINTS].RelIndexNextPoint := 0;
END_METHOD

END_FUNCTION_BLOCK

// ---- GlobalTextList.TcGTLO
TEXTLIST GlobalTextList
  580 = 'As Soon As Possible'
  179 = 'Change Mode'
  999 = 'Change Table'
  530 = 'Current Table: %d'
  527 = 'Instant'
  67 = 'Instantaneous'
  368 = 'Next Cycle'
  75 = 'NextCycle'
END_TEXTLIST

// ---- VISUs/Visualization.TcVIS
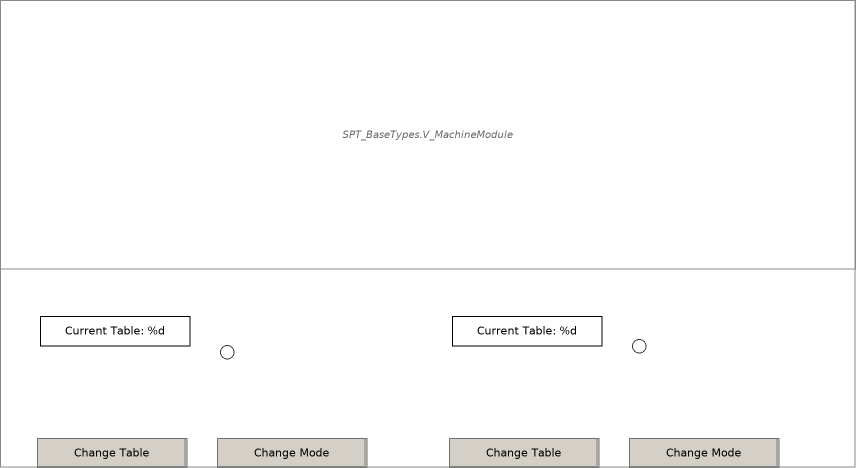
VISUALIZATION Visualization  // 856x468
    Frame (0,0 856x269)
        shows SPT_BaseTypes.V_MachineModule(HMI := MAIN.Machine.PackMLBaseModule_HMI)
    Button (37,438 150x30), "Change Table"
        toggle MAIN.Machine.CamModule_TableSelect.HMI.Cmd.ChangeTable
    Rectangle (40,316 150x30), "Current Table: %d", text variable: MAIN.Machine.CamModule_TableSelect.HMI.Sts.CurrentTable
    RadioButton (218,296 150x112), variable: MAIN.Machine.CamModule_TableSelect.HMI.Cfg.CamActivationMode
        Areas[0]: Text=Instantaneous
        Areas[1]: Text=Next Cycle
        Areas[2]: Text=As Soon As Possible
    Button (217,438 150x30), "Change Mode"
        toggle MAIN.Machine.CamModule_TableSelect.HMI.Cmd.ChangeMode
    Button (449,438 150x30), "Change Table"
        toggle MAIN.Machine.CamModule_UpdateTable.HMI.Cmd.ChangeTable
    Rectangle (452,316 150x30), "Current Table: %d", text variable: MAIN.Machine.CamModule_UpdateTable.HMI.Sts.CurrentTable
    RadioButton (630,296 150x100), variable: MAIN.Machine.CamModule_UpdateTable.HMI.Cfg.CamActivationMode
        Areas[0]: Text=Instantaneous
        Areas[1]: Text=Next Cycle
        Areas[2]: Text=As Soon As Possible
    Button (629,438 150x30), "Change Mode"
        toggle MAIN.Machine.CamModule_UpdateTable.HMI.Cmd.ChangeMode
END_VISUALIZATION
